{attribute 'GeneratedUsingTerminal: EL5101--0000'}
{attribute addProperty BoxType "EL5101--0000"}
{attribute addProperty Id "StatusAT %I*USINT1ValueAT %I*UINT2LatchAT %I*UINT2"}
{attribute addProperty CRC "3104192441"}
{attribute addProperty Size "5"}
TYPE Channel_B90637B9 EXTENDS InputBase_8311D824 :
STRUCT
	{attribute addProperty Name "Status"}
	Status AT %I* : USINT;
	{attribute addProperty Name "Value"}
	Value AT %I* : UINT;
	{attribute addProperty Name "Latch"}
	Latch AT %I* : UINT;
END_STRUCT
END_TYPE

(* stored: Version 1.2.0.0, ProductVersion 3.1.4024.9
   DUT Channel_B90637B9: Id {56c71af6-580f-448d-a69a-7d1c10066210} *)
